FUNCTION_BLOCK FB_EdgeMonitor
VAR_INPUT
END_VAR
VAR_OUTPUT
END_VAR
VAR
	fTrig : F_TRIG;
	rTrig : R_TRIG;
END_VAR

METHOD FallingEdge : BOOL
VAR_INPUT
	i_SignalToMonitor : BOOL;
END_VAR
fTrig(CLK := i_SignalToMonitor);
IF fTrig.Q THEN
	FallingEdge := TRUE;
ELSE
	FallingEdge := FALSE;
END_IF
END_METHOD

END_FUNCTION_BLOCK

(* stored: Version 1.1.0.1, ProductVersion 3.1.4024.12
   POU FB_EdgeMonitor: Id {b4f4b128-6ea1-4c4d-a2da-8452d09a25cd}, SpecialFunc None
   Method FallingEdge: Id {9f6860f0-86f9-48da-acd9-800852b1e36b} *)
